// TIA Portal V17 export
// export: Created 2025-03-07T09:19:00.9335589Z, ExportSetting WithDefaults, DisplayName Totally Integrated Automation Portal, DisplayVersion V17 Update 8, DisplayName TIA Portal Openness, DisplayVersion V17 Update 8, DisplayName TIA Portal Version Control Interface, DisplayVersion V17, DisplayName SINAMICS Startdrive Advanced, DisplayVersion V17 SP2, DisplayName SINAMICS Startdrive G110M, G120, G120C, G120D, G120P, G115D, DisplayVersion V17 SP2, DisplayName SINAMICS Startdrive G130, G150, S120, S150, SINAMICS MV, S210, DisplayVersion V17 SP2, DisplayName STEP 7 Professional, DisplayVersion V17 Update 8, DisplayName SINUMERIK ONE STEP 7 Toolbox, DisplayVersion V17 Update 12, DisplayName SINUMERIK 840D sl STEP 7 Toolbox, DisplayVersion V17 Update 12, DisplayName STEP 7 Safety, DisplayVersion V17 Update 6, DisplayName WinCC Advanced, DisplayVersion V17 Update 8
DATA_BLOCK "DB16207_METHODCALL_U01_STA3_MEAS_RESET_TRIGGER"   // DB16207
// stored: AutoNumber false, DBAccessibleFromOPCUA true, DBAccessibleFromWebserver true, InstanceOfName OPC_UA_MethodCall_C, OfSystemLibElement OPC_UA_MethodCall_C, OfSystemLibVersion 1.0
"OPC_UA_MethodCall_C"
   // VAR_INPUT
   //    REQ : Bool;
   //    MaintainSession : Bool;
   //    ServerEndpointUrl : String[254];
   //    SessionConnectInfo : OPC_UA_SessionConnectInfo;
   //    NamespaceUrisCount : UInt;
   //    MethodHdlCount : UInt;
   //    MethodHdl : DWord;
   // END_VAR
   // VAR_OUTPUT
   //    Done : Bool;
   //    Busy : Bool;
   //    Error : Bool;
   //    Status : DWord;
   // END_VAR
   // VAR_IN_OUT
   //    NamespaceUris : Variant;
   //    NamespaceStatusList : Variant;
   //    NamespaceIndexes : Variant;
   //    ObjectNodeIDs : Variant;
   //    MethodNodeIDs : Variant;
   //    MethodHdls : Variant;
   //    StatusList : Variant;
   //    MethodResult : Variant;
   //    InputArguments : Variant;
   //    OutputArguments : Variant;
   // END_VAR
   // VAR
   //    s_OPC_UA_Connect_Instance { ExternalAccessible := 'False'; ExternalVisible := 'False'; ExternalWritable := 'False'; S7_SetPoint := 'True'} : OPC_UA_Connect;
   //    s_OPC_UA_NamespaceGetIndexList_Instance { ExternalAccessible := 'False'; ExternalVisible := 'False'; ExternalWritable := 'False'; S7_SetPoint := 'True'} : OPC_UA_NamespaceGetIndexList;
   //    s_OPC_UA_MethodGetHandleList_Instance { ExternalAccessible := 'False'; ExternalVisible := 'False'; ExternalWritable := 'False'; S7_SetPoint := 'True'} : OPC_UA_MethodGetHandleList;
   //    s_OPC_UA_MethodCall_Instance { ExternalAccessible := 'False'; ExternalVisible := 'False'; ExternalWritable := 'False'; S7_SetPoint := 'True'} : OPC_UA_MethodCall;
   //    s_OPC_UA_MethodReleaseHandleList_Instance { ExternalAccessible := 'False'; ExternalVisible := 'False'; ExternalWritable := 'False'; S7_SetPoint := 'True'} : OPC_UA_MethodReleaseHandleList;
   //    s_OPC_UA_Disconnect_Instance { ExternalAccessible := 'False'; ExternalVisible := 'False'; ExternalWritable := 'False'; S7_SetPoint := 'True'} : OPC_UA_Disconnect;
   //    s_OPC_UA_ConnectionGetStatus_Instance { ExternalAccessible := 'False'; ExternalVisible := 'False'; ExternalWritable := 'False'; S7_SetPoint := 'True'} : OPC_UA_ConnectionGetStatus;
   //    s_BlockState { ExternalAccessible := 'False'; ExternalVisible := 'False'; ExternalWritable := 'False'} : Struct
   //       CurrentState { ExternalAccessible := 'False'; ExternalVisible := 'False'; ExternalWritable := 'False'} : Word;
   //       NextState { ExternalAccessible := 'False'; ExternalVisible := 'False'; ExternalWritable := 'False'} : Word;
   //       ErrorState { ExternalAccessible := 'False'; ExternalVisible := 'False'; ExternalWritable := 'False'} : Word;
   //       PrevState { ExternalAccessible := 'False'; ExternalVisible := 'False'; ExternalWritable := 'False'} : Word;
   //    END_STRUCT;
   //    s_ConnectionHdl { ExternalAccessible := 'False'; ExternalVisible := 'False'; ExternalWritable := 'False'} : DWord;
   //    s_LastStatusError { ExternalAccessible := 'False'; ExternalVisible := 'False'; ExternalWritable := 'False'} : DWord;
   //    s_LastSubStateWithError { ExternalAccessible := 'False'; ExternalVisible := 'False'; ExternalWritable := 'False'} : Word;
   //    s_StatusList_CurrentElement { ExternalAccessible := 'False'; ExternalVisible := 'False'; ExternalWritable := 'False'} : UDInt;
   //    s_ReconnectTimer { ExternalAccessible := 'False'; ExternalVisible := 'False'; ExternalWritable := 'False'; S7_SetPoint := 'True'} : TON_TIME;
   // END_VAR
BEGIN
END_DATA_BLOCK
